TYPE S_Drive_control_settings :
STRUCT
	Max_drive_speed:INT;
	Max_drive_torque:INT;
	Speed_S_func_scans:INT;
	Current_S_func_scans:INT;
	No_start_time:TIME;
	Motor_fed_delay:TIME;
	Stall_time:TIME;
	Stall_speed:INT;
	Torque_ctrl_max_speed:INT;
	Brake_apply_speed:INT;
	Trail_brake_speed:INT;
	De_energise_to_trail:BOOL;
	Single_lever_control:BOOL;
	Stall_current:INT;
	Backout_min_speed:INT;

	(*Torque prediction settings*)	
	Lh_cage_mass_current:REAL;
	Rh_cage_mass_current:REAL;
	Lh_rope_mass_current:REAL;
	Rh_rope_mass_current:REAL;
	Full_payload_current:REAL;
	A_s2_per_m:REAL;
	Accel_torque_lag:TIME;
	Dynamic_friction_current:REAL;

END_STRUCT
END_TYPE

(* stored: Version 1.1.0.1, ProductVersion 3.1.4024.0
   DUT S_Drive_control_settings: Id {77fb175a-f626-42bc-8ab4-2d99c8d4b0b9} *)
